Fanuc KAREL source: kx00020.KL

-- PROVISIONAL review KL for V940-1; original PC SHA256 34344bdcf1574aa7fce948845f9d9c8d222620dd66edda4e0343442dc231b642
-- Incomplete behavior may be omitted. Consult companion uncertainty JSON. Do not deploy.
PROGRAM KX00020
%NOLOCKGROUP
BEGIN
  -- V9_ZERO_TABLE_METADATA_HINT layout=0001; no indexed target words; source/name/runtime held
  -- UNRESOLVED_PC offsets 5-17; opcodes 3F,22,9D,33,61
  -- UNRESOLVED_PC offsets 22-37; opcodes 22,9D,33,5E,75
  -- UNRESOLVED_PC offsets 42-46; opcodes 7F
END KX00020
